# EPICS substitutions: PIP-II/RFPI2/rfpi-fdr-sw-mgmt-ioc-main/ina-managementApp/Db/general.substitutions
file general.template {
pattern{ acc, sys, group, num }
{ PIP2IT, pHB650, RFPI, ina}
}
